FUNCTION_BLOCK ConcatStringRpcHandler IMPLEMENTS I_RpcHandler
VAR
END_VAR

METHOD Handle
VAR_INPUT
	Parameters : I_Deserializer;
	Response : I_SynchronousRpcResponse;
END_VAR
VAR
	str1 : T_MAXSTRING;
	str2 : T_MAXSTRING;
	result : T_MAXSTRING;
END_VAR
IF NOT Parameters.TryGetKeyString('STR1',str1) THEN
	Response.RejectWithMessage('Missing STR1 parameter');
	RETURN;
END_IF

IF NOT Parameters.TryGetKeyString('STR2',str2) THEN
	Response.RejectWithMessage('Missing STR2 parameter');
	RETURN;
END_IF

result := CONCAT(str1, str2);
Response.CompleteWithString(result);
END_METHOD

END_FUNCTION_BLOCK

(* stored: Version 1.1.0.1, ProductVersion 3.1.4024.12
   POU ConcatStringRpcHandler: Id {6b570563-90ca-0168-02e7-bdb7639403ed}, SpecialFunc None
   Method Handle: Id {c47d4b37-7d63-0cb6-0d96-0ea952bbbe7f} *)
